% RSLogix 500 project Practise-6.RSS, saved by version 8.30.00.16 %
PROJECT "UNTITLED"    % processor: MicroLogix 1000 %

PROGRAM FILES
  LAD 2 "MAIN_PROG"  6 rungs
  LAD 3 "USER_FAULT"  1 rungs
  LAD 4 "HSC_INT"  1 rungs
  LAD 5 "STI_INT"  1 rungs
  LAD 6, 7, 8, 9, 10, 11, 12, 13, 14, 15, 16: only END

DATA FILES
  O0 OUTPUT  1 elements
  I1 INPUT  2 elements
  S2 STATUS  33 elements
  B3 BINARY  32 elements
  T4 TIMER  40 elements
  C5 COUNTER  32 elements
  R6 CONTROL  16 elements
  N7 INTEGER  105 elements

LADDER 2 "MAIN_PROG"
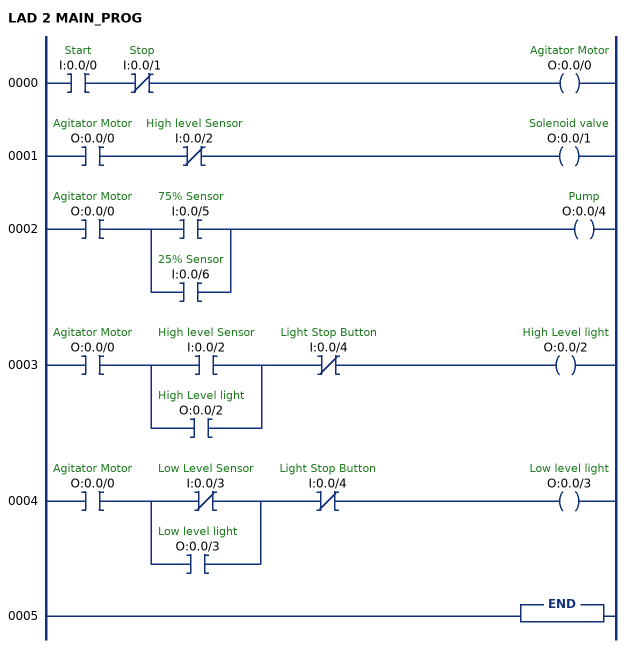
% Rung: 0 %
SOR XIC I:0.0/0 XIO I:0.0/1 OTE O:0.0/0 EOR
%   I:0.0/0  "Start" %
%   I:0.0/1  "Stop" %
%   O:0.0/0  "Agitator Motor" %
% Rung: 1 %
SOR XIC O:0.0/0 XIO I:0.0/2 OTE O:0.0/1 EOR
%   O:0.0/0  "Agitator Motor" %
%   I:0.0/2  "High level Sensor" %
%   O:0.0/1  "Solenoid valve" %
% Rung: 2 %
SOR XIC O:0.0/0 BST XIC I:0.0/5 NXB XIC I:0.0/6 BND OTE O:0.0/4 EOR
%   O:0.0/0  "Agitator Motor" %
%   I:0.0/5  "75% Sensor" %
%   I:0.0/6  "25% Sensor" %
%   O:0.0/4  "Pump" %
% Rung: 3 %
SOR XIC O:0.0/0 BST XIC I:0.0/2 NXB XIC O:0.0/2 BND XIO I:0.0/4 OTE O:0.0/2 EOR
%   O:0.0/0  "Agitator Motor" %
%   I:0.0/2  "High level Sensor" %
%   O:0.0/2  "High Level light" %
%   I:0.0/4  "Light Stop Button" %
% Rung: 4 %
SOR XIC O:0.0/0 BST XIO I:0.0/3 NXB XIC O:0.0/3 BND XIO I:0.0/4 OTE O:0.0/3 EOR
%   O:0.0/0  "Agitator Motor" %
%   I:0.0/3  "Low Level Sensor" %
%   O:0.0/3  "Low level light" %
%   I:0.0/4  "Light Stop Button" %
% Rung: 5 %
SOR END EOR
